// TIA Portal V18 export
DATA_BLOCK "testing_purposes"   // DB2
{ S7_Optimized_Access := 'TRUE' }
VERSION : 0.1
// stored: AutoNumber true, DBAccessibleFromOPCUA true, IsOnlyStoredInLoadMemory false, IsRetainMemResEnabled false, IsWriteProtectedInAS false, MemoryReserve 100
   VAR
      emc_calculated : Real;   // EMC_returned
      Temperature : Real := 20.0;   // Chamber temperature [C]
      Air_humi : Real;   // Air humidity [%]
      TemperatureWet : Real := 15.0;   // Wet bulb temperature [C]
      Air_humi_calc : Real;   // Calculated air humidity [%]
      TemperatureWet_calc : Real;   // Calculated wet bulb temperature [C]
      real_sig : Real := 0.0;
      real_win_len : UInt := 20;
      filt_real_sig : Real;
      real_ret_result : Int;   // Real filter work result
      lreal_sig : Real := 0.0;
      lreal_win_len : UInt := 30;
      filt_lreal_sig : Real;
      lreal_ret_result : Int;   // lReal filter work result
   END_VAR
BEGIN
END_DATA_BLOCK
